FUNCTION_BLOCK L3_SetupRouterM (* Basic Function Block Type *)
  (* Standard: 61499-2 *)
  (* Version 0.0, 2014-11-19, 4DIAC-IDE, 4DIAC-Consortium *)
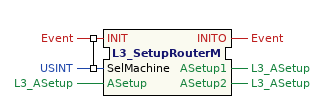
  EVENT_INPUT
    INIT WITH SelMachine;
  END_EVENT
  EVENT_OUTPUT
    INITO;
  END_EVENT
  VAR_INPUT
    SelMachine : USINT; (* Routing condition *)
  END_VAR
  SOCKETS
    ASetup : L3_ASetup;
  END_SOCKETS
  PLUGS
    ASetup1 : L3_ASetup;
    ASetup2 : L3_ASetup;
  END_PLUGS
  VAR
    i : USINT; (* loop variable *)
    Select : BOOL; (* Routing condition *)
  END_VAR
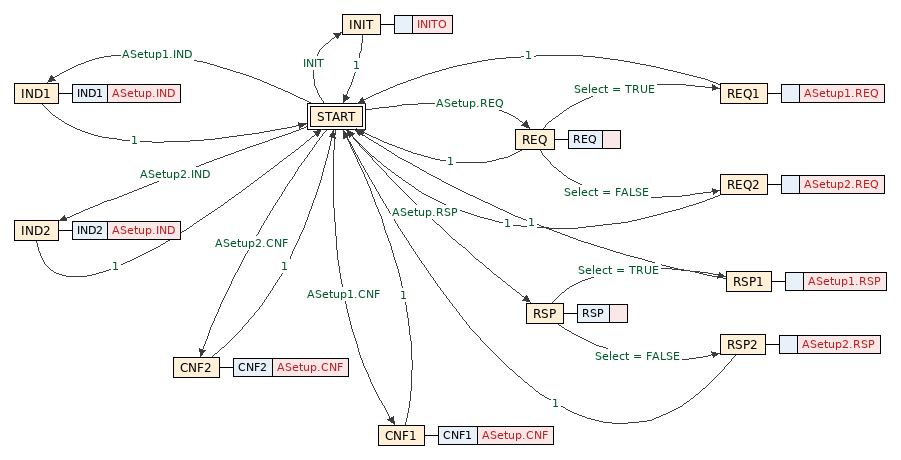
  EC_STATES
    START; (* Initial State *)
    REQ : REQ; (* Normal execution *)
    INIT : -> INITO;
    REQ1 : -> ASetup1.REQ;
    REQ2 : -> ASetup2.REQ;
    RSP : RSP;
    RSP1 : -> ASetup1.RSP;
    RSP2 : -> ASetup2.RSP;
    CNF1 : CNF1 -> ASetup.CNF;
    CNF2 : CNF2 -> ASetup.CNF;
    IND1 : IND1 -> ASetup.IND;
    IND2 : IND2 -> ASetup.IND;
  END_STATES
  EC_TRANSITIONS
    START TO REQ := ASetup.REQ;
    REQ TO START := 1;
    START TO INIT := INIT;
    INIT TO START := 1;
    REQ TO REQ1 := Select = TRUE;
    REQ TO REQ2 := Select = FALSE;
    REQ1 TO START := 1;
    REQ2 TO START := 1;
    START TO RSP := ASetup.RSP;
    RSP TO RSP1 := Select = TRUE;
    RSP TO RSP2 := Select = FALSE;
    RSP1 TO START := 1;
    RSP2 TO START := 1;
    START TO IND1 := ASetup1.IND;
    IND1 TO START := 1;
    START TO IND2 := ASetup2.IND;
    IND2 TO START := 1;
    START TO CNF2 := ASetup2.CNF;
    CNF2 TO START := 1;
    START TO CNF1 := ASetup1.CNF;
    CNF1 TO START := 1;
  END_TRANSITIONS
  ALGORITHM REQ IN ST: (* Normally executed algorithm *)
IF ASetup.MID = SelMachine THEN
	Select := TRUE;
	FOR i:=0 TO 2 DO
		ASetup1.PartInfoP[i] :=ASetup.PartInfoP[i];
	END_FOR;
	ASetup1.MID := ASetup.MID;
	FOR i:=0 TO 19 DO
		ASetup1.OPIDS[i] := ASetup.OPIDS[i];
		ASetup1.OPParams[i] := ASetup.OPParams[i];
	END_FOR;
	ASetup1.Fixture := ASetup.Fixture;
ELSE
	Select := FALSE;
	FOR i:=0 TO 2 DO
		ASetup2.PartInfoP[i] :=ASetup.PartInfoP[i];
	END_FOR;
	ASetup2.MID := ASetup.MID;
	FOR i:=0 TO 19 DO
		ASetup2.OPIDS[i] := ASetup.OPIDS[i];
		ASetup2.OPParams[i] := ASetup.OPParams[i];
	END_FOR;
	ASetup2.Fixture := ASetup.Fixture;
END_IF;
  END_ALGORITHM
  ALGORITHM RSP IN ST: (* new algorithm *)
IF ASetup.MID = SelMachine THEN
	Select := TRUE;
	ASetup1.MID := ASetup.MID;
ELSE
	Select := FALSE;
	ASetup2.MID := ASetup.MID;
END_IF;
  END_ALGORITHM
  ALGORITHM CNF1 IN ST: (* new algorithm *)
ASetup.PartInfoS[0] := ASetup1.PartInfoS[0];
ASetup.PartInfoS[1] := ASetup1.PartInfoS[1];
ASetup.PartInfoS[2] := ASetup1.PartInfoS[2];
  END_ALGORITHM
  ALGORITHM CNF2 IN ST: (* new algorithm *)
ASetup.PartInfoS[0] := ASetup2.PartInfoS[0];
ASetup.PartInfoS[1] := ASetup2.PartInfoS[1];
ASetup.PartInfoS[2] := ASetup2.PartInfoS[2];
  END_ALGORITHM
  ALGORITHM IND1 IN ST: (* new algorithm *)
ASetup.PartInfoS[0] := ASetup1.PartInfoS[0];
ASetup.PartInfoS[1] := ASetup1.PartInfoS[1];
ASetup.PartInfoS[2] := ASetup1.PartInfoS[2];
ASetup.ENDID := ASetup1.ENDID;
  END_ALGORITHM
  ALGORITHM IND2 IN ST: (* new algorithm *)
ASetup.PartInfoS[0] := ASetup2.PartInfoS[0];
ASetup.PartInfoS[1] := ASetup2.PartInfoS[1];
ASetup.PartInfoS[2] := ASetup2.PartInfoS[2];
ASetup.ENDID := ASetup2.ENDID;
  END_ALGORITHM
END_FUNCTION_BLOCK
